(* CoDeSys 2.3 export: PROC_ERR_DIG_OUTS.EXP *)

(* POU 60_Error handling/Process Errors/proc_Err_DIG_outs, ST *)
PROGRAM proc_Err_DIG_outs
VAR

END_VAR
;
END_PROGRAM
